REGION Network 51: Step[690] : JOB[6] Step End
   RUNG wire#powerrail
      { S7_Templates := "SrcType := DInt" } EQ_Contact(in1 := "Unit1.Em4.ControlNodes".sideTapeFixStage.sequence.status.currentStep, in2 := #JOB_6_STEP_90)
      Contact( "Unit1.Em4.ControlNodes".sideTapeFixStage.sequence.status.seqActive )
      wire#w1
      Coil( "Unit1.Em4.ControlNodes".sideTapeFixStage."step".action1[690] )
   END_RUNG
   RUNG wire#w1
      Coil( "Unit1.Em4.ControlNodes".sideTapeFixStage."step".transition1[690] )
   END_RUNG
   RUNG wire#w1
      Contact( "Unit1.Em4.ControlNodes".sideTapeFixStage."step".transition1[690] )
      { S7_Templates := "time_type := Time" } #statTonTime[690].TON(pt := T#100ms, et =>)
      Move(in := #STEP_IDLE, out1 => "Unit1.Em4.ControlNodes".sideTapeFixStage.sequence.status.nextStep)
   END_RUNG
   // the same network as SCL:
   "Unit1.Em4.ControlNodes".sideTapeFixStage."step".action1[690] := ("Unit1.Em4.ControlNodes".sideTapeFixStage.sequence.status.currentStep = #JOB_6_STEP_90) AND "Unit1.Em4.ControlNodes".sideTapeFixStage.sequence.status.seqActive;
   "Unit1.Em4.ControlNodes".sideTapeFixStage."step".transition1[690] := ("Unit1.Em4.ControlNodes".sideTapeFixStage.sequence.status.currentStep = #JOB_6_STEP_90) AND "Unit1.Em4.ControlNodes".sideTapeFixStage.sequence.status.seqActive;
   #statTonTime[690].TON(IN := ("Unit1.Em4.ControlNodes".sideTapeFixStage.sequence.status.currentStep = #JOB_6_STEP_90) AND "Unit1.Em4.ControlNodes".sideTapeFixStage.sequence.status.seqActive AND "Unit1.Em4.ControlNodes".sideTapeFixStage."step".transition1[690],
                         PT := T#100ms);
   IF #statTonTime[690].Q THEN
       "Unit1.Em4.ControlNodes".sideTapeFixStage.sequence.status.nextStep := #STEP_IDLE;
   END_IF;
END_REGION

REGION Network 52: *************** JOB[7] JR PUT=AUTO *************************
END_REGION

REGION Network 53: Step[701] : JOB[7] Condition
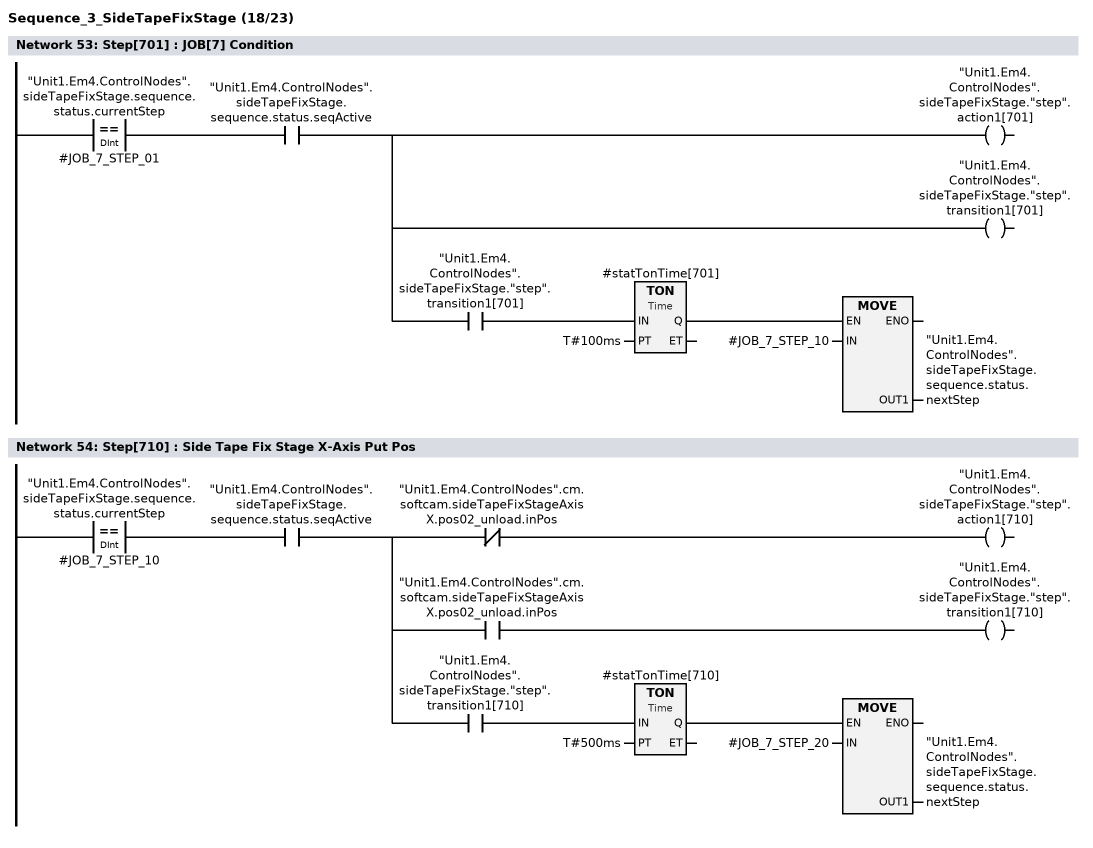
   RUNG wire#powerrail
      { S7_Templates := "SrcType := DInt" } EQ_Contact(in1 := "Unit1.Em4.ControlNodes".sideTapeFixStage.sequence.status.currentStep, in2 := #JOB_7_STEP_01)
      Contact( "Unit1.Em4.ControlNodes".sideTapeFixStage.sequence.status.seqActive )
      wire#w1
      Coil( "Unit1.Em4.ControlNodes".sideTapeFixStage."step".action1[701] )
   END_RUNG
   RUNG wire#w1
      Coil( "Unit1.Em4.ControlNodes".sideTapeFixStage."step".transition1[701] )
   END_RUNG
   RUNG wire#w1
      Contact( "Unit1.Em4.ControlNodes".sideTapeFixStage."step".transition1[701] )
      { S7_Templates := "time_type := Time" } #statTonTime[701].TON(pt := T#100ms, et =>)
      Move(in := #JOB_7_STEP_10, out1 => "Unit1.Em4.ControlNodes".sideTapeFixStage.sequence.status.nextStep)
   END_RUNG
   // the same network as SCL:
   "Unit1.Em4.ControlNodes".sideTapeFixStage."step".action1[701] := ("Unit1.Em4.ControlNodes".sideTapeFixStage.sequence.status.currentStep = #JOB_7_STEP_01) AND "Unit1.Em4.ControlNodes".sideTapeFixStage.sequence.status.seqActive;
   "Unit1.Em4.ControlNodes".sideTapeFixStage."step".transition1[701] := ("Unit1.Em4.ControlNodes".sideTapeFixStage.sequence.status.currentStep = #JOB_7_STEP_01) AND "Unit1.Em4.ControlNodes".sideTapeFixStage.sequence.status.seqActive;
   #statTonTime[701].TON(IN := ("Unit1.Em4.ControlNodes".sideTapeFixStage.sequence.status.currentStep = #JOB_7_STEP_01) AND "Unit1.Em4.ControlNodes".sideTapeFixStage.sequence.status.seqActive AND "Unit1.Em4.ControlNodes".sideTapeFixStage."step".transition1[701],
                         PT := T#100ms);
   IF #statTonTime[701].Q THEN
       "Unit1.Em4.ControlNodes".sideTapeFixStage.sequence.status.nextStep := #JOB_7_STEP_10;
   END_IF;
END_REGION

REGION Network 54: Step[710] : Side Tape Fix Stage X-Axis Put Pos
   RUNG wire#powerrail
      { S7_Templates := "SrcType := DInt" } EQ_Contact(in1 := "Unit1.Em4.ControlNodes".sideTapeFixStage.sequence.status.currentStep, in2 := #JOB_7_STEP_10)
      Contact( "Unit1.Em4.ControlNodes".sideTapeFixStage.sequence.status.seqActive )
      wire#w1
      I_Contact( "Unit1.Em4.ControlNodes".cm.softcam.sideTapeFixStageAxisX.pos02_unload.inPos )
      Coil( "Unit1.Em4.ControlNodes".sideTapeFixStage."step".action1[710] )
   END_RUNG
   RUNG wire#w1
      Contact( "Unit1.Em4.ControlNodes".cm.softcam.sideTapeFixStageAxisX.pos02_unload.inPos )
      Coil( "Unit1.Em4.ControlNodes".sideTapeFixStage."step".transition1[710] )
   END_RUNG
   RUNG wire#w1
      Contact( "Unit1.Em4.ControlNodes".sideTapeFixStage."step".transition1[710] )
      { S7_Templates := "time_type := Time" } #statTonTime[710].TON(pt := T#500ms, et =>)
      Move(in := #JOB_7_STEP_20, out1 => "Unit1.Em4.ControlNodes".sideTapeFixStage.sequence.status.nextStep)
   END_RUNG
   // the same network as SCL:
   #_w1 := ("Unit1.Em4.ControlNodes".sideTapeFixStage.sequence.status.currentStep = #JOB_7_STEP_10) AND "Unit1.Em4.ControlNodes".sideTapeFixStage.sequence.status.seqActive;
   "Unit1.Em4.ControlNodes".sideTapeFixStage."step".action1[710] := #_w1 AND NOT "Unit1.Em4.ControlNodes".cm.softcam.sideTapeFixStageAxisX.pos02_unload.inPos;
   "Unit1.Em4.ControlNodes".sideTapeFixStage."step".transition1[710] := #_w1 AND "Unit1.Em4.ControlNodes".cm.softcam.sideTapeFixStageAxisX.pos02_unload.inPos;
   #statTonTime[710].TON(IN := #_w1 AND "Unit1.Em4.ControlNodes".sideTapeFixStage."step".transition1[710],
                         PT := T#500ms);
   IF #statTonTime[710].Q THEN
       "Unit1.Em4.ControlNodes".sideTapeFixStage.sequence.status.nextStep := #JOB_7_STEP_20;
   END_IF;
END_REGION

REGION Network 55: Step[720] : Side Tape Fix Stage [Unloading Request] => Transfer PP Left
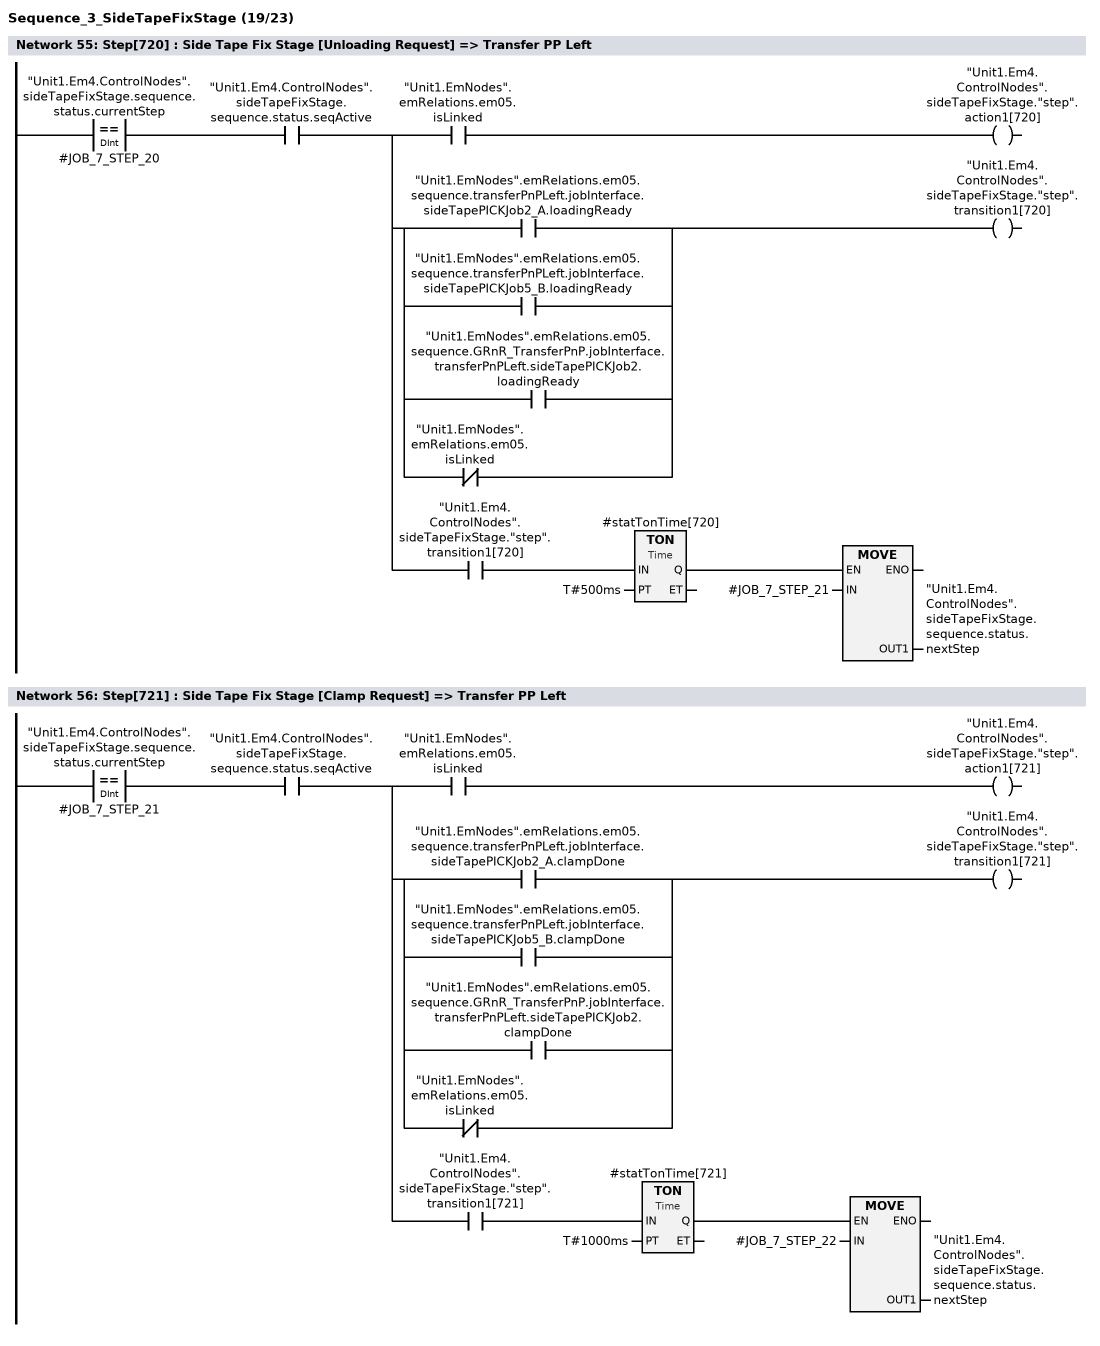
   RUNG wire#powerrail
      { S7_Templates := "SrcType := DInt" } EQ_Contact(in1 := "Unit1.Em4.ControlNodes".sideTapeFixStage.sequence.status.currentStep, in2 := #JOB_7_STEP_20)
      Contact( "Unit1.Em4.ControlNodes".sideTapeFixStage.sequence.status.seqActive )
      wire#w1
      Contact( "Unit1.EmNodes".emRelations.em05.isLinked )
      Coil( "Unit1.Em4.ControlNodes".sideTapeFixStage."step".action1[720] )
   END_RUNG
   RUNG wire#w1
      Contact( "Unit1.EmNodes".emRelations.em05.sequence.transferPnPLeft.jobInterface.sideTapePICKJob2_A.loadingReady )
      wire#w2
      Coil( "Unit1.Em4.ControlNodes".sideTapeFixStage."step".transition1[720] )
   END_RUNG
   RUNG wire#w1
      Contact( "Unit1.EmNodes".emRelations.em05.sequence.transferPnPLeft.jobInterface.sideTapePICKJob5_B.loadingReady )
   END_RUNG wire#w2
   RUNG wire#w1
      Contact( "Unit1.EmNodes".emRelations.em05.sequence.GRnR_TransferPnP.jobInterface.transferPnPLeft.sideTapePICKJob2.loadingReady )
   END_RUNG wire#w2
   RUNG wire#w1
      I_Contact( "Unit1.EmNodes".emRelations.em05.isLinked )
   END_RUNG wire#w2
   RUNG wire#w1
      Contact( "Unit1.Em4.ControlNodes".sideTapeFixStage."step".transition1[720] )
      { S7_Templates := "time_type := Time" } #statTonTime[720].TON(pt := T#500ms, et =>)
      Move(in := #JOB_7_STEP_21, out1 => "Unit1.Em4.ControlNodes".sideTapeFixStage.sequence.status.nextStep)
   END_RUNG
   // the same network as SCL:
   #_w1 := ("Unit1.Em4.ControlNodes".sideTapeFixStage.sequence.status.currentStep = #JOB_7_STEP_20) AND "Unit1.Em4.ControlNodes".sideTapeFixStage.sequence.status.seqActive;
   "Unit1.Em4.ControlNodes".sideTapeFixStage."step".action1[720] := #_w1 AND "Unit1.EmNodes".emRelations.em05.isLinked;
   "Unit1.Em4.ControlNodes".sideTapeFixStage."step".transition1[720] := #_w1 AND ("Unit1.EmNodes".emRelations.em05.sequence.transferPnPLeft.jobInterface.sideTapePICKJob2_A.loadingReady OR "Unit1.EmNodes".emRelations.em05.sequence.transferPnPLeft.jobInterface.sideTapePICKJob5_B.loadingReady OR "Unit1.EmNodes".emRelations.em05.sequence.GRnR_TransferPnP.jobInterface.transferPnPLeft.sideTapePICKJob2.loadingReady OR NOT "Unit1.EmNodes".emRelations.em05.isLinked);
   #statTonTime[720].TON(IN := #_w1 AND "Unit1.Em4.ControlNodes".sideTapeFixStage."step".transition1[720],
                         PT := T#500ms);
   IF #statTonTime[720].Q THEN
       "Unit1.Em4.ControlNodes".sideTapeFixStage.sequence.status.nextStep := #JOB_7_STEP_21;
   END_IF;
END_REGION

REGION Network 56: Step[721] : Side Tape Fix Stage [Clamp Request] => Transfer PP Left
   RUNG wire#powerrail
      { S7_Templates := "SrcType := DInt" } EQ_Contact(in1 := "Unit1.Em4.ControlNodes".sideTapeFixStage.sequence.status.currentStep, in2 := #JOB_7_STEP_21)
      Contact( "Unit1.Em4.ControlNodes".sideTapeFixStage.sequence.status.seqActive )
      wire#w1
      Contact( "Unit1.EmNodes".emRelations.em05.isLinked )
      Coil( "Unit1.Em4.ControlNodes".sideTapeFixStage."step".action1[721] )
   END_RUNG
   RUNG wire#w1
      Contact( "Unit1.EmNodes".emRelations.em05.sequence.transferPnPLeft.jobInterface.sideTapePICKJob2_A.clampDone )
      wire#w2
      Coil( "Unit1.Em4.ControlNodes".sideTapeFixStage."step".transition1[721] )
   END_RUNG
   RUNG wire#w1
      Contact( "Unit1.EmNodes".emRelations.em05.sequence.transferPnPLeft.jobInterface.sideTapePICKJob5_B.clampDone )
   END_RUNG wire#w2
   RUNG wire#w1
      Contact( "Unit1.EmNodes".emRelations.em05.sequence.GRnR_TransferPnP.jobInterface.transferPnPLeft.sideTapePICKJob2.clampDone )
   END_RUNG wire#w2
   RUNG wire#w1
      I_Contact( "Unit1.EmNodes".emRelations.em05.isLinked )
   END_RUNG wire#w2
   RUNG wire#w1
      Contact( "Unit1.Em4.ControlNodes".sideTapeFixStage."step".transition1[721] )
      { S7_Templates := "time_type := Time" } #statTonTime[721].TON(pt := T#1000ms, et =>)
      Move(in := #JOB_7_STEP_22, out1 => "Unit1.Em4.ControlNodes".sideTapeFixStage.sequence.status.nextStep)
   END_RUNG
   // the same network as SCL:
   #_w1 := ("Unit1.Em4.ControlNodes".sideTapeFixStage.sequence.status.currentStep = #JOB_7_STEP_21) AND "Unit1.Em4.ControlNodes".sideTapeFixStage.sequence.status.seqActive;
   "Unit1.Em4.ControlNodes".sideTapeFixStage."step".action1[721] := #_w1 AND "Unit1.EmNodes".emRelations.em05.isLinked;
   "Unit1.Em4.ControlNodes".sideTapeFixStage."step".transition1[721] := #_w1 AND ("Unit1.EmNodes".emRelations.em05.sequence.transferPnPLeft.jobInterface.sideTapePICKJob2_A.clampDone OR "Unit1.EmNodes".emRelations.em05.sequence.transferPnPLeft.jobInterface.sideTapePICKJob5_B.clampDone OR "Unit1.EmNodes".emRelations.em05.sequence.GRnR_TransferPnP.jobInterface.transferPnPLeft.sideTapePICKJob2.clampDone OR NOT "Unit1.EmNodes".emRelations.em05.isLinked);
   #statTonTime[721].TON(IN := #_w1 AND "Unit1.Em4.ControlNodes".sideTapeFixStage."step".transition1[721],
                         PT := T#1000ms);
   IF #statTonTime[721].Q THEN
       "Unit1.Em4.ControlNodes".sideTapeFixStage.sequence.status.nextStep := #JOB_7_STEP_22;
   END_IF;
END_REGION

REGION Network 57: Step[722] : Side Tape Fix Stage Clamp Open
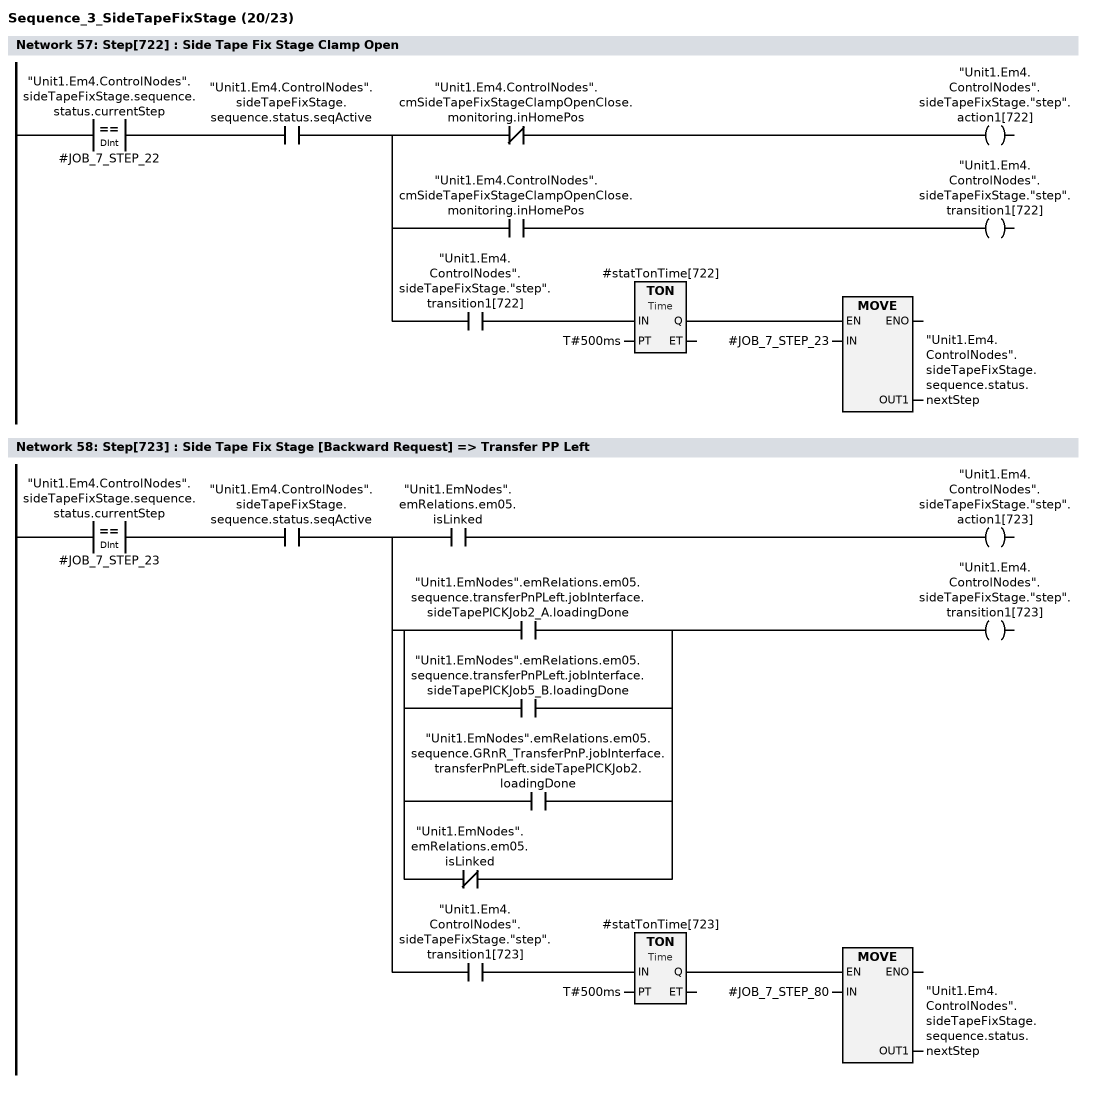
   RUNG wire#powerrail
      { S7_Templates := "SrcType := DInt" } EQ_Contact(in1 := "Unit1.Em4.ControlNodes".sideTapeFixStage.sequence.status.currentStep, in2 := #JOB_7_STEP_22)
      Contact( "Unit1.Em4.ControlNodes".sideTapeFixStage.sequence.status.seqActive )
      wire#w1
      I_Contact( "Unit1.Em4.ControlNodes".cmSideTapeFixStageClampOpenClose.monitoring.inHomePos )
      Coil( "Unit1.Em4.ControlNodes".sideTapeFixStage."step".action1[722] )
   END_RUNG
   RUNG wire#w1
      Contact( "Unit1.Em4.ControlNodes".cmSideTapeFixStageClampOpenClose.monitoring.inHomePos )
      Coil( "Unit1.Em4.ControlNodes".sideTapeFixStage."step".transition1[722] )
   END_RUNG
   RUNG wire#w1
      Contact( "Unit1.Em4.ControlNodes".sideTapeFixStage."step".transition1[722] )
      { S7_Templates := "time_type := Time" } #statTonTime[722].TON(pt := T#500ms, et =>)
      Move(in := #JOB_7_STEP_23, out1 => "Unit1.Em4.ControlNodes".sideTapeFixStage.sequence.status.nextStep)
   END_RUNG
   // the same network as SCL:
   #_w1 := ("Unit1.Em4.ControlNodes".sideTapeFixStage.sequence.status.currentStep = #JOB_7_STEP_22) AND "Unit1.Em4.ControlNodes".sideTapeFixStage.sequence.status.seqActive;
   "Unit1.Em4.ControlNodes".sideTapeFixStage."step".action1[722] := #_w1 AND NOT "Unit1.Em4.ControlNodes".cmSideTapeFixStageClampOpenClose.monitoring.inHomePos;
   "Unit1.Em4.ControlNodes".sideTapeFixStage."step".transition1[722] := #_w1 AND "Unit1.Em4.ControlNodes".cmSideTapeFixStageClampOpenClose.monitoring.inHomePos;
   #statTonTime[722].TON(IN := #_w1 AND "Unit1.Em4.ControlNodes".sideTapeFixStage."step".transition1[722],
                         PT := T#500ms);
   IF #statTonTime[722].Q THEN
       "Unit1.Em4.ControlNodes".sideTapeFixStage.sequence.status.nextStep := #JOB_7_STEP_23;
   END_IF;
END_REGION

REGION Network 58: Step[723] : Side Tape Fix Stage [Backward Request] => Transfer PP Left
   RUNG wire#powerrail
      { S7_Templates := "SrcType := DInt" } EQ_Contact(in1 := "Unit1.Em4.ControlNodes".sideTapeFixStage.sequence.status.currentStep, in2 := #JOB_7_STEP_23)
      Contact( "Unit1.Em4.ControlNodes".sideTapeFixStage.sequence.status.seqActive )
      wire#w1
      Contact( "Unit1.EmNodes".emRelations.em05.isLinked )
      Coil( "Unit1.Em4.ControlNodes".sideTapeFixStage."step".action1[723] )
   END_RUNG
   RUNG wire#w1
      Contact( "Unit1.EmNodes".emRelations.em05.sequence.transferPnPLeft.jobInterface.sideTapePICKJob2_A.loadingDone )
      wire#w2
      Coil( "Unit1.Em4.ControlNodes".sideTapeFixStage."step".transition1[723] )
   END_RUNG
   RUNG wire#w1
      Contact( "Unit1.EmNodes".emRelations.em05.sequence.transferPnPLeft.jobInterface.sideTapePICKJob5_B.loadingDone )
   END_RUNG wire#w2
   RUNG wire#w1
      Contact( "Unit1.EmNodes".emRelations.em05.sequence.GRnR_TransferPnP.jobInterface.transferPnPLeft.sideTapePICKJob2.loadingDone )
   END_RUNG wire#w2
   RUNG wire#w1
      I_Contact( "Unit1.EmNodes".emRelations.em05.isLinked )
   END_RUNG wire#w2
   RUNG wire#w1
      Contact( "Unit1.Em4.ControlNodes".sideTapeFixStage."step".transition1[723] )
      { S7_Templates := "time_type := Time" } #statTonTime[723].TON(pt := T#500ms, et =>)
      Move(in := #JOB_7_STEP_80, out1 => "Unit1.Em4.ControlNodes".sideTapeFixStage.sequence.status.nextStep)
   END_RUNG
   // the same network as SCL:
   #_w1 := ("Unit1.Em4.ControlNodes".sideTapeFixStage.sequence.status.currentStep = #JOB_7_STEP_23) AND "Unit1.Em4.ControlNodes".sideTapeFixStage.sequence.status.seqActive;
   "Unit1.Em4.ControlNodes".sideTapeFixStage."step".action1[723] := #_w1 AND "Unit1.EmNodes".emRelations.em05.isLinked;
   "Unit1.Em4.ControlNodes".sideTapeFixStage."step".transition1[723] := #_w1 AND ("Unit1.EmNodes".emRelations.em05.sequence.transferPnPLeft.jobInterface.sideTapePICKJob2_A.loadingDone OR "Unit1.EmNodes".emRelations.em05.sequence.transferPnPLeft.jobInterface.sideTapePICKJob5_B.loadingDone OR "Unit1.EmNodes".emRelations.em05.sequence.GRnR_TransferPnP.jobInterface.transferPnPLeft.sideTapePICKJob2.loadingDone OR NOT "Unit1.EmNodes".emRelations.em05.isLinked);
   #statTonTime[723].TON(IN := #_w1 AND "Unit1.Em4.ControlNodes".sideTapeFixStage."step".transition1[723],
                         PT := T#500ms);
   IF #statTonTime[723].Q THEN
       "Unit1.Em4.ControlNodes".sideTapeFixStage.sequence.status.nextStep := #JOB_7_STEP_80;
   END_IF;
END_REGION

REGION Network 59: Step[780] : Side Tape Fix Stage X-Axis Wait Pos
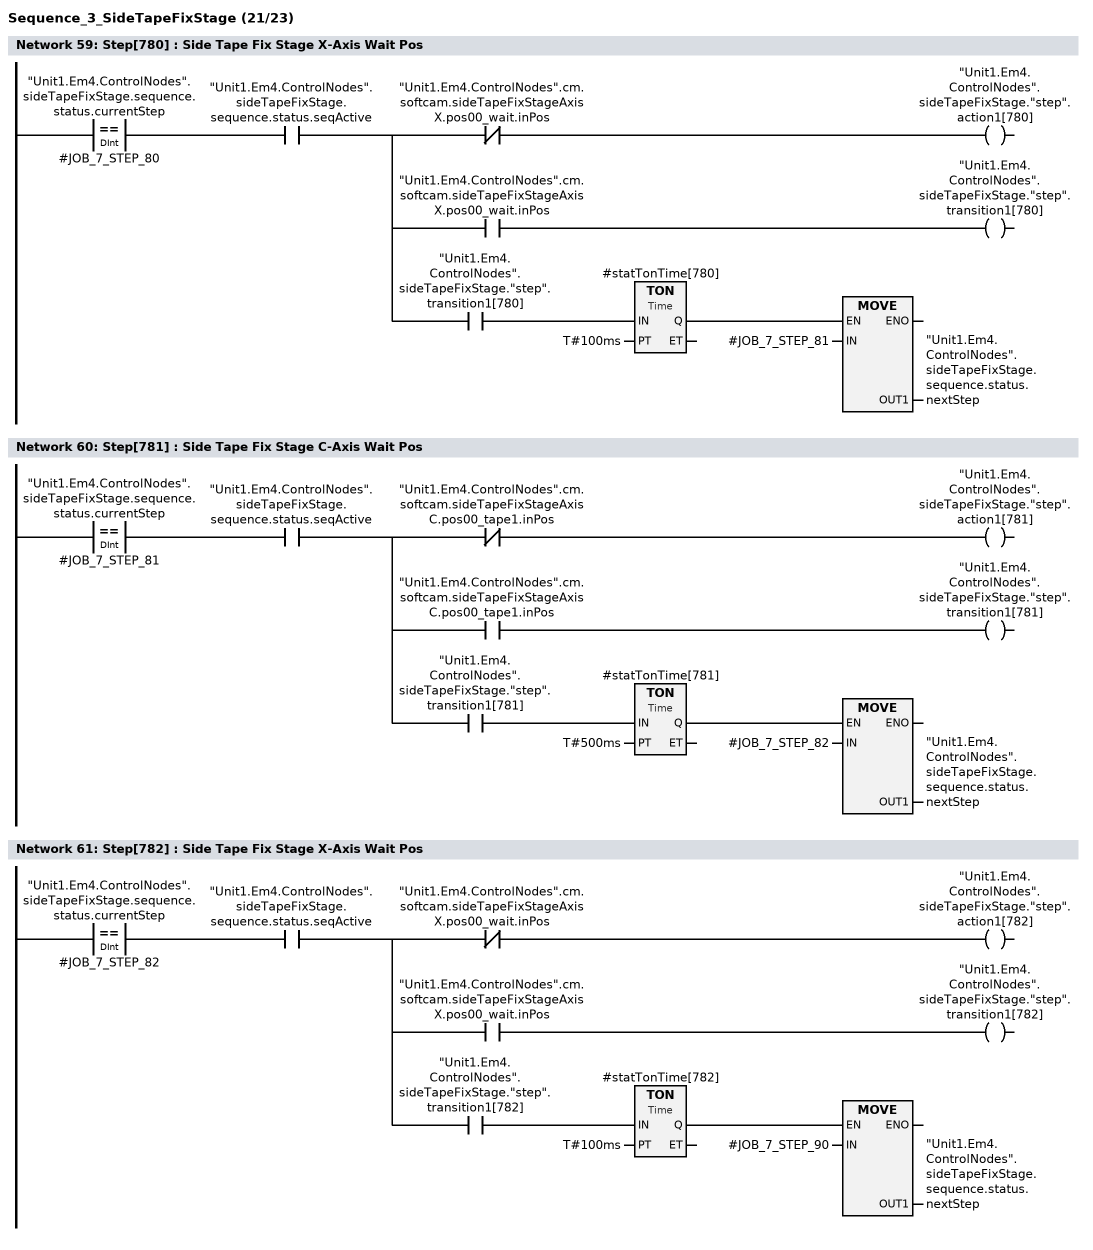
   RUNG wire#powerrail
      { S7_Templates := "SrcType := DInt" } EQ_Contact(in1 := "Unit1.Em4.ControlNodes".sideTapeFixStage.sequence.status.currentStep, in2 := #JOB_7_STEP_80)
      Contact( "Unit1.Em4.ControlNodes".sideTapeFixStage.sequence.status.seqActive )
      wire#w1
      I_Contact( "Unit1.Em4.ControlNodes".cm.softcam.sideTapeFixStageAxisX.pos00_wait.inPos )
      Coil( "Unit1.Em4.ControlNodes".sideTapeFixStage."step".action1[780] )
   END_RUNG
   RUNG wire#w1
      Contact( "Unit1.Em4.ControlNodes".cm.softcam.sideTapeFixStageAxisX.pos00_wait.inPos )
      Coil( "Unit1.Em4.ControlNodes".sideTapeFixStage."step".transition1[780] )
   END_RUNG
   RUNG wire#w1
      Contact( "Unit1.Em4.ControlNodes".sideTapeFixStage."step".transition1[780] )
      { S7_Templates := "time_type := Time" } #statTonTime[780].TON(pt := T#100ms, et =>)
      Move(in := #JOB_7_STEP_81, out1 => "Unit1.Em4.ControlNodes".sideTapeFixStage.sequence.status.nextStep)
   END_RUNG
   // the same network as SCL:
   #_w1 := ("Unit1.Em4.ControlNodes".sideTapeFixStage.sequence.status.currentStep = #JOB_7_STEP_80) AND "Unit1.Em4.ControlNodes".sideTapeFixStage.sequence.status.seqActive;
   "Unit1.Em4.ControlNodes".sideTapeFixStage."step".action1[780] := #_w1 AND NOT "Unit1.Em4.ControlNodes".cm.softcam.sideTapeFixStageAxisX.pos00_wait.inPos;
   "Unit1.Em4.ControlNodes".sideTapeFixStage."step".transition1[780] := #_w1 AND "Unit1.Em4.ControlNodes".cm.softcam.sideTapeFixStageAxisX.pos00_wait.inPos;
   #statTonTime[780].TON(IN := #_w1 AND "Unit1.Em4.ControlNodes".sideTapeFixStage."step".transition1[780],
                         PT := T#100ms);
   IF #statTonTime[780].Q THEN
       "Unit1.Em4.ControlNodes".sideTapeFixStage.sequence.status.nextStep := #JOB_7_STEP_81;
   END_IF;
END_REGION

REGION Network 60: Step[781] : Side Tape Fix Stage C-Axis Wait Pos
   RUNG wire#powerrail
      { S7_Templates := "SrcType := DInt" } EQ_Contact(in1 := "Unit1.Em4.ControlNodes".sideTapeFixStage.sequence.status.currentStep, in2 := #JOB_7_STEP_81)
      Contact( "Unit1.Em4.ControlNodes".sideTapeFixStage.sequence.status.seqActive )
      wire#w1
      I_Contact( "Unit1.Em4.ControlNodes".cm.softcam.sideTapeFixStageAxisC.pos00_tape1.inPos )
      Coil( "Unit1.Em4.ControlNodes".sideTapeFixStage."step".action1[781] )
   END_RUNG
   RUNG wire#w1
      Contact( "Unit1.Em4.ControlNodes".cm.softcam.sideTapeFixStageAxisC.pos00_tape1.inPos )
      Coil( "Unit1.Em4.ControlNodes".sideTapeFixStage."step".transition1[781] )
   END_RUNG
   RUNG wire#w1
      Contact( "Unit1.Em4.ControlNodes".sideTapeFixStage."step".transition1[781] )
      { S7_Templates := "time_type := Time" } #statTonTime[781].TON(pt := T#500ms, et =>)
      Move(in := #JOB_7_STEP_82, out1 => "Unit1.Em4.ControlNodes".sideTapeFixStage.sequence.status.nextStep)
   END_RUNG
   // the same network as SCL:
   #_w1 := ("Unit1.Em4.ControlNodes".sideTapeFixStage.sequence.status.currentStep = #JOB_7_STEP_81) AND "Unit1.Em4.ControlNodes".sideTapeFixStage.sequence.status.seqActive;
   "Unit1.Em4.ControlNodes".sideTapeFixStage."step".action1[781] := #_w1 AND NOT "Unit1.Em4.ControlNodes".cm.softcam.sideTapeFixStageAxisC.pos00_tape1.inPos;
   "Unit1.Em4.ControlNodes".sideTapeFixStage."step".transition1[781] := #_w1 AND "Unit1.Em4.ControlNodes".cm.softcam.sideTapeFixStageAxisC.pos00_tape1.inPos;
   #statTonTime[781].TON(IN := #_w1 AND "Unit1.Em4.ControlNodes".sideTapeFixStage."step".transition1[781],
                         PT := T#500ms);
   IF #statTonTime[781].Q THEN
       "Unit1.Em4.ControlNodes".sideTapeFixStage.sequence.status.nextStep := #JOB_7_STEP_82;
   END_IF;
END_REGION

REGION Network 61: Step[782] : Side Tape Fix Stage X-Axis Wait Pos
   RUNG wire#powerrail
      { S7_Templates := "SrcType := DInt" } EQ_Contact(in1 := "Unit1.Em4.ControlNodes".sideTapeFixStage.sequence.status.currentStep, in2 := #JOB_7_STEP_82)
      Contact( "Unit1.Em4.ControlNodes".sideTapeFixStage.sequence.status.seqActive )
      wire#w1
      I_Contact( "Unit1.Em4.ControlNodes".cm.softcam.sideTapeFixStageAxisX.pos00_wait.inPos )
      Coil( "Unit1.Em4.ControlNodes".sideTapeFixStage."step".action1[782] )
   END_RUNG
   RUNG wire#w1
      Contact( "Unit1.Em4.ControlNodes".cm.softcam.sideTapeFixStageAxisX.pos00_wait.inPos )
      Coil( "Unit1.Em4.ControlNodes".sideTapeFixStage."step".transition1[782] )
   END_RUNG
   RUNG wire#w1
      Contact( "Unit1.Em4.ControlNodes".sideTapeFixStage."step".transition1[782] )
      { S7_Templates := "time_type := Time" } #statTonTime[782].TON(pt := T#100ms, et =>)
      Move(in := #JOB_7_STEP_90, out1 => "Unit1.Em4.ControlNodes".sideTapeFixStage.sequence.status.nextStep)
   END_RUNG
   // the same network as SCL:
   #_w1 := ("Unit1.Em4.ControlNodes".sideTapeFixStage.sequence.status.currentStep = #JOB_7_STEP_82) AND "Unit1.Em4.ControlNodes".sideTapeFixStage.sequence.status.seqActive;
   "Unit1.Em4.ControlNodes".sideTapeFixStage."step".action1[782] := #_w1 AND NOT "Unit1.Em4.ControlNodes".cm.softcam.sideTapeFixStageAxisX.pos00_wait.inPos;
   "Unit1.Em4.ControlNodes".sideTapeFixStage."step".transition1[782] := #_w1 AND "Unit1.Em4.ControlNodes".cm.softcam.sideTapeFixStageAxisX.pos00_wait.inPos;
   #statTonTime[782].TON(IN := #_w1 AND "Unit1.Em4.ControlNodes".sideTapeFixStage."step".transition1[782],
                         PT := T#100ms);
   IF #statTonTime[782].Q THEN
       "Unit1.Em4.ControlNodes".sideTapeFixStage.sequence.status.nextStep := #JOB_7_STEP_90;
   END_IF;
END_REGION

REGION Network 62: Step[790] : JOB[7] Step End
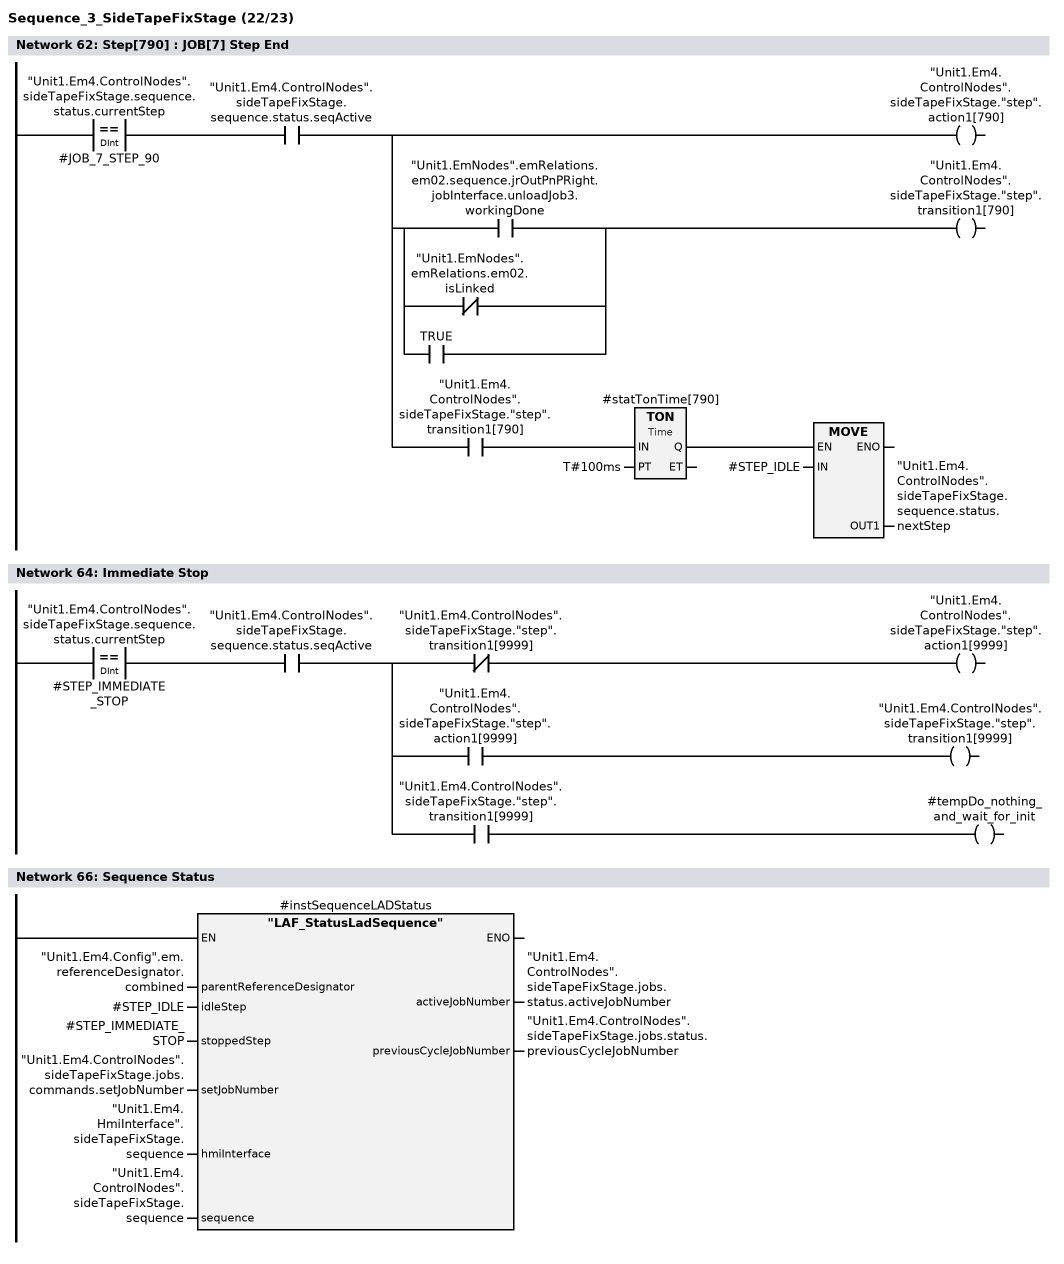
   RUNG wire#powerrail
      { S7_Templates := "SrcType := DInt" } EQ_Contact(in1 := "Unit1.Em4.ControlNodes".sideTapeFixStage.sequence.status.currentStep, in2 := #JOB_7_STEP_90)
      Contact( "Unit1.Em4.ControlNodes".sideTapeFixStage.sequence.status.seqActive )
      wire#w1
      Coil( "Unit1.Em4.ControlNodes".sideTapeFixStage."step".action1[790] )
   END_RUNG
   RUNG wire#w1
      Contact( "Unit1.EmNodes".emRelations.em02.sequence.jrOutPnPRight.jobInterface.unloadJob3.workingDone )
      wire#w2
      Coil( "Unit1.Em4.ControlNodes".sideTapeFixStage."step".transition1[790] )
   END_RUNG
   RUNG wire#w1
      I_Contact( "Unit1.EmNodes".emRelations.em02.isLinked )
   END_RUNG wire#w2
   RUNG wire#w1
      Contact( TRUE )
   END_RUNG wire#w2
   RUNG wire#w1
      Contact( "Unit1.Em4.ControlNodes".sideTapeFixStage."step".transition1[790] )
      { S7_Templates := "time_type := Time" } #statTonTime[790].TON(pt := T#100ms, et =>)
      Move(in := #STEP_IDLE, out1 => "Unit1.Em4.ControlNodes".sideTapeFixStage.sequence.status.nextStep)
   END_RUNG
   // the same network as SCL:
   "Unit1.Em4.ControlNodes".sideTapeFixStage."step".action1[790] := ("Unit1.Em4.ControlNodes".sideTapeFixStage.sequence.status.currentStep = #JOB_7_STEP_90) AND "Unit1.Em4.ControlNodes".sideTapeFixStage.sequence.status.seqActive;
   "Unit1.Em4.ControlNodes".sideTapeFixStage."step".transition1[790] := ("Unit1.Em4.ControlNodes".sideTapeFixStage.sequence.status.currentStep = #JOB_7_STEP_90) AND "Unit1.Em4.ControlNodes".sideTapeFixStage.sequence.status.seqActive AND ("Unit1.EmNodes".emRelations.em02.sequence.jrOutPnPRight.jobInterface.unloadJob3.workingDone OR NOT "Unit1.EmNodes".emRelations.em02.isLinked OR TRUE);
   #statTonTime[790].TON(IN := ("Unit1.Em4.ControlNodes".sideTapeFixStage.sequence.status.currentStep = #JOB_7_STEP_90) AND "Unit1.Em4.ControlNodes".sideTapeFixStage.sequence.status.seqActive AND "Unit1.Em4.ControlNodes".sideTapeFixStage."step".transition1[790],
                         PT := T#100ms);
   IF #statTonTime[790].Q THEN
       "Unit1.Em4.ControlNodes".sideTapeFixStage.sequence.status.nextStep := #STEP_IDLE;
   END_IF;
END_REGION

REGION Network 63: *************** IMMEDIATE STOP ****************
END_REGION

REGION Network 64: Immediate Stop
   RUNG wire#powerrail
      { S7_Templates := "SrcType := DInt" } EQ_Contact(in1 := "Unit1.Em4.ControlNodes".sideTapeFixStage.sequence.status.currentStep, in2 := #STEP_IMMEDIATE_STOP)
      Contact( "Unit1.Em4.ControlNodes".sideTapeFixStage.sequence.status.seqActive )
      wire#w1
      I_Contact( "Unit1.Em4.ControlNodes".sideTapeFixStage."step".transition1[9999] )
      Coil( "Unit1.Em4.ControlNodes".sideTapeFixStage."step".action1[9999] )
   END_RUNG
   RUNG wire#w1
      Contact( "Unit1.Em4.ControlNodes".sideTapeFixStage."step".action1[9999] )
      Coil( "Unit1.Em4.ControlNodes".sideTapeFixStage."step".transition1[9999] )
   END_RUNG
   RUNG wire#w1
      Contact( "Unit1.Em4.ControlNodes".sideTapeFixStage."step".transition1[9999] )
      Coil( #tempDo_nothing_and_wait_for_init )
   END_RUNG
   // the same network as SCL:
   #_w1 := ("Unit1.Em4.ControlNodes".sideTapeFixStage.sequence.status.currentStep = #STEP_IMMEDIATE_STOP) AND "Unit1.Em4.ControlNodes".sideTapeFixStage.sequence.status.seqActive;
   "Unit1.Em4.ControlNodes".sideTapeFixStage."step".action1[9999] := #_w1 AND NOT "Unit1.Em4.ControlNodes".sideTapeFixStage."step".transition1[9999];
   "Unit1.Em4.ControlNodes".sideTapeFixStage."step".transition1[9999] := #_w1 AND "Unit1.Em4.ControlNodes".sideTapeFixStage."step".action1[9999];
   #tempDo_nothing_and_wait_for_init := #_w1 AND "Unit1.Em4.ControlNodes".sideTapeFixStage."step".transition1[9999];
END_REGION

REGION Network 65: *************** STATUS **********************
END_REGION

REGION Network 66: Sequence Status
   RUNG wire#powerrail
      #instSequenceLADStatus(parentReferenceDesignator := "Unit1.Em4.Config".em.referenceDesignator.combined, idleStep := #STEP_IDLE, stoppedStep := #STEP_IMMEDIATE_STOP, setJobNumber := "Unit1.Em4.ControlNodes".sideTapeFixStage.jobs.commands.setJobNumber, hmiInterface := "Unit1.Em4.HmiInterface".sideTapeFixStage.sequence, sequence := "Unit1.Em4.ControlNodes".sideTapeFixStage.sequence, activeJobNumber => "Unit1.Em4.ControlNodes".sideTapeFixStage.jobs.status.activeJobNumber, previousCycleJobNumber => "Unit1.Em4.ControlNodes".sideTapeFixStage.jobs.status.previousCycleJobNumber)
   END_RUNG
   // the same network as SCL:
   #instSequenceLADStatus(parentReferenceDesignator := "Unit1.Em4.Config".em.referenceDesignator.combined,   // "LAF_StatusLadSequence"
                          idleStep := #STEP_IDLE,
                          stoppedStep := #STEP_IMMEDIATE_STOP,
                          setJobNumber := "Unit1.Em4.ControlNodes".sideTapeFixStage.jobs.commands.setJobNumber,
                          hmiInterface := "Unit1.Em4.HmiInterface".sideTapeFixStage.sequence,
                          sequence := "Unit1.Em4.ControlNodes".sideTapeFixStage.sequence,
                          activeJobNumber => "Unit1.Em4.ControlNodes".sideTapeFixStage.jobs.status.activeJobNumber,
                          previousCycleJobNumber => "Unit1.Em4.ControlNodes".sideTapeFixStage.jobs.status.previousCycleJobNumber);
END_REGION

REGION Network 67: Update Job History
   // Update the History of jobs if a new job was started
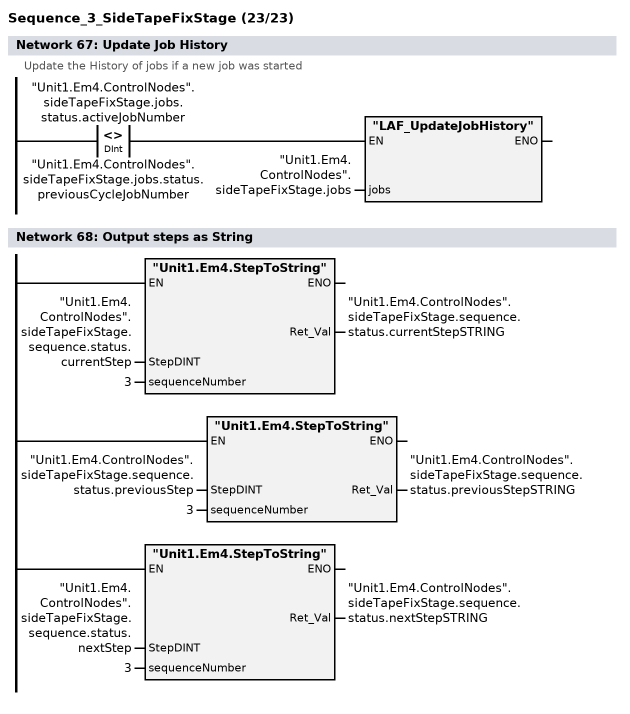
   RUNG wire#powerrail
      { S7_Templates := "SrcType := DInt" } NE_Contact(in1 := "Unit1.Em4.ControlNodes".sideTapeFixStage.jobs.status.activeJobNumber, in2 := "Unit1.Em4.ControlNodes".sideTapeFixStage.jobs.status.previousCycleJobNumber)
      "LAF_UpdateJobHistory"(jobs := "Unit1.Em4.ControlNodes".sideTapeFixStage.jobs)
   END_RUNG
   // the same network as SCL:
   IF "Unit1.Em4.ControlNodes".sideTapeFixStage.jobs.status.activeJobNumber <> "Unit1.Em4.ControlNodes".sideTapeFixStage.jobs.status.previousCycleJobNumber THEN
       "LAF_UpdateJobHistory"(jobs := "Unit1.Em4.ControlNodes".sideTapeFixStage.jobs);
   END_IF;
END_REGION

REGION Network 68: Output steps as String
   RUNG wire#powerrail
      "Unit1.Em4.StepToString"(StepDINT := "Unit1.Em4.ControlNodes".sideTapeFixStage.sequence.status.currentStep, sequenceNumber := 3, Ret_Val => "Unit1.Em4.ControlNodes".sideTapeFixStage.sequence.status.currentStepSTRING)
   END_RUNG
   RUNG wire#powerrail
      "Unit1.Em4.StepToString"(StepDINT := "Unit1.Em4.ControlNodes".sideTapeFixStage.sequence.status.previousStep, sequenceNumber := 3, Ret_Val => "Unit1.Em4.ControlNodes".sideTapeFixStage.sequence.status.previousStepSTRING)
   END_RUNG
   RUNG wire#powerrail
      "Unit1.Em4.StepToString"(StepDINT := "Unit1.Em4.ControlNodes".sideTapeFixStage.sequence.status.nextStep, sequenceNumber := 3, Ret_Val => "Unit1.Em4.ControlNodes".sideTapeFixStage.sequence.status.nextStepSTRING)
   END_RUNG
   // the same network as SCL:
   "Unit1.Em4.ControlNodes".sideTapeFixStage.sequence.status.currentStepSTRING := "Unit1.Em4.StepToString"(StepDINT := "Unit1.Em4.ControlNodes".sideTapeFixStage.sequence.status.currentStep,
                           sequenceNumber := 3);
   "Unit1.Em4.ControlNodes".sideTapeFixStage.sequence.status.previousStepSTRING := "Unit1.Em4.StepToString"(StepDINT := "Unit1.Em4.ControlNodes".sideTapeFixStage.sequence.status.previousStep,
                           sequenceNumber := 3);
   "Unit1.Em4.ControlNodes".sideTapeFixStage.sequence.status.nextStepSTRING := "Unit1.Em4.StepToString"(StepDINT := "Unit1.Em4.ControlNodes".sideTapeFixStage.sequence.status.nextStep,
                           sequenceNumber := 3);
END_REGION
END_FUNCTION_BLOCK
